TYPE ZData :
STRUCT
  Config : ZDataConfig;
  Machine : ZDataMachine;
  Calibration : ZDataCalibration;
  Recipe : ZDataRecipe;
END_STRUCT
END_TYPE

(* stored: Version 1.1.0.1
   DUT ZData: Id {006e9cd1-1b1d-49a9-bb3c-0a597740c897} *)
